FUNCTION_BLOCK Stage17 (* Template for a Basic Function Block Type *)
  (* Standard: 61499-2 *)
  (* Version 1.0, 2021-06-20, HP *)
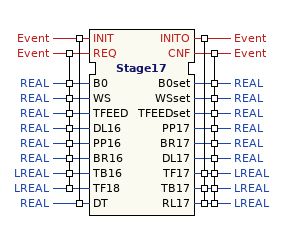
  EVENT_INPUT
    INIT WITH DT; (* Initialization Request *)
    REQ WITH B0, WS, TFEED, DL16, PP16, BR16, TB16, TF18; (* Normal Execution Request *)
  END_EVENT
  EVENT_OUTPUT
    INITO WITH TB17, RL17, TF17; (* Initialization Confirm *)
    CNF WITH TB17, DL17, TF17, BR17, PP17, TFEEDset, B0set, WSset, RL17; (* Execution Confirmation *)
  END_EVENT
  VAR_INPUT
    B0 : REAL;
    WS : REAL;
    TFEED : REAL;
    DL16 : REAL;
    PP16 : REAL;
    BR16 : REAL;
    TB16 : LREAL;
    TF18 : LREAL;
    DT : REAL;
  END_VAR
  VAR_OUTPUT
    B0set : REAL;
    WSset : REAL;
    TFEEDset : REAL;
    PP17 : REAL;
    BR17 : REAL;
    DL17 : REAL;
    TF17 : LREAL;
    TB17 : LREAL;
    RL17 : LREAL;
  END_VAR
  VAR
    AB : REAL; (* internal variabel *)
    UU : REAL;
    TREF : REAL;
    AD : REAL;
    AHC : REAL;
    AHR : REAL;
    AS : REAL;
    REC : REAL;
    WN : REAL;
    WN_1 : REAL;
    XKN : REAL;
    C1 : REAL;
    HS : REAL;
    G : REAL;
    W1 : REAL;
    TFREC : REAL;
    TS : REAL;
    DTS : REAL;
    TF17_last : REAL;
    RL17_last : REAL;
    TB17_last : REAL;
    USS : REAL;
    RHOB : REAL;
    CPB : REAL;
    CPF : REAL;
    FMW : REAL;
    HLV : REAL;
    HV : REAL;
    BPR : REAL;
    FMC : REAL;
    U : REAL;
    A : REAL;
    B : REAL;
    C : REAL;
    D1 : REAL;
    d : REAL;
    a : REAL;
    A1 : REAL;
    A2 : REAL;
    A3 : REAL;
    A4 : REAL;
    A5 : REAL;
    A6 : REAL;
    p : REAL;
    q : REAL;
    TC : REAL;
    PC : REAL;
    DTB17 : REAL;
    DEN17 : REAL;
    DH17 : REAL;
    DP17 : REAL;
    DPDH17 : REAL;
    DT17 : REAL;
    m : REAL;
    n : REAL;
    VR17 : REAL;
    DELTA17 : REAL;
    DELTA39 : REAL;
    DELTA61 : REAL;
    DELTA17_last : REAL;
    DELTA39_last : REAL;
    DELTA61_last : REAL;
  END_VAR
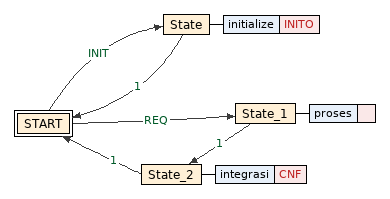
  EC_STATES
    START; (* Initial State *)
    State : initialize -> INITO;
    State_1 : proses;
    State_2 : integrasi -> CNF;
  END_STATES
  EC_TRANSITIONS
    START TO State := INIT;
    State TO START := 1;
    START TO State_1 := REQ;
    State_1 TO State_2 := 1;
    State_2 TO START := 1;
  END_TRANSITIONS
  ALGORITHM initialize IN ST: (* Initialization algorithm *)
TREF :=273.15;
AB :=57.2727;
AHC :=4069.2;
AHR :=2639.7;
AS :=3225.7;
REC :=0.0;
//TF2:=TF2;

//TFEED :=TFEED1+TREF;
 //TS:=TS1+TREF;
WN :=3.0;
XKN :=0.68;
HS:=0.11;
G :=9.81;
W1 :=0.50;

RL17 := 0.613640754894074;
TB17 := 323.552719861124;
TF17 := 320.275377684374;
TF18 := 318.266914942048;


RL17_last :=RL17;
TB17_last :=TB17;
TF17_last :=TF17;
  END_ALGORITHM
  ALGORITHM proses IN ST: (* kalkulasi *)
UU := TFEED;
U :=UU;

USS :=49.767;
C1 :=0.625;
RHOB :=1032.4; //maassa jenis brine
CPB :=1.00; //heatcapacity Brine
CPF :=1.00; //heat capacity feed
FMW :=23654.0;
HLV :=563.7959;
HV :=625.1971;
BPR :=2.192;
FMC :=34736.09;
//U :=UU; //feed temp



///  Calculate the physical properties

//A :=3.2437814;
//B :=5.86826*0.001;
//C :=1.1702379*0.00000001;
//D1 :=2.1878462*0.001;
//TC :=647.27;
//PC :=218.167;


A1 :=3.2437814;
A2:=5.86826*0.001;
A3:=1.1702379*0.00000001;
A4 :=2.1878462*0.001;
A5 :=647.27;
A6 :=218.167;

DTB17 :=A5-TB17;
DEN17 :=(A1+A2*DTB17+A3*DTB17*DTB17*DTB17)/(1+A4*DTB17)*DTB17/TB17;
p:=DEN17;
q:=10.0;
PP17 :=A6/(EXPT(q, p));

// calculate the brine flow rates
DP17:=PP16-PP17;
DH17:=RL17-C1*HS;
DPDH17 :=DP17*101000+G*RHOB*DH17;
m:=DPDH17*RHOB;
n:=0.5;
BR17 :=WN*XKN*RL17*(EXPT(m, n));
BR17 :=BR17*60.0/1000.0;

// calculate the vapor flow rates

DT17 :=TB17-BPR/1.8-(TF18+TF17)*0.5;
VR17:=U*AHC*DT17/HLV/1000.0;
DL17 :=DL16+VR17;


//// state equation
DELTA17 :=(BR16-BR17-VR17)*1000.0/RHOB/AB;
DELTA39 :=((BR16*CPB*(TB16-TB17))-VR17*(HV-CPB*(TB17-TREF)))*1000.0/AB/RHOB/CPB/RL17;
DELTA61 :=(B0*CPF*(TF18-TF17)*1000+(U*AHC*DT17))/FMW/CPF;
  END_ALGORITHM
  ALGORITHM integrasi IN ST: (* new algorithm *)
B0set:=B0;
WSset:=WS ;
TFEEDset:=TFEED;
//integrasi
RL17 := (DELTA17 + DELTA17_last)*0.5*DT + RL17_last;
DELTA17_last :=DELTA17 ;
RL17_last :=RL17;

TB17:= (DELTA39 + DELTA39_last)*0.5*DT + TB17_last;
DELTA39_last :=DELTA39 ;
TB17_last:=TB17;

TF17 := (DELTA61 + DELTA61_last)*0.5*DT + TF17_last;
DELTA61_last :=DELTA61 ;
TF17_last :=TF17;
  END_ALGORITHM
END_FUNCTION_BLOCK
